// TIA Portal V20 export
DATA_BLOCK "LPFE_TelemetryKVPData"   // DB252
// stored: Access Published, MemoryReserve 100, Namespace PFE
   VAR
      TelemetryStructData : "LPFE_typeTelemetryContent";
   END_VAR
BEGIN
END_DATA_BLOCK
